FUNCTION_BLOCK FB_AUT_MODIFY EXTENDS FB_AUT_ABSTRACT
    (****************************************************************************)
    (*	POU_AUT_zxx			Bausteinaufrufe Station	zxx							*)
    (*	Status				ungetestet											*)
    (*  Version:			1.0													*)
    (*	Beschrieb:																*)
    (*																			*)
    (*	Abläufe:			FB_ABLzxxA		Hauptablauf							*)
    (*																			*)
    (*																			*)
    (* 	25.09.2019/Dj															*)
    (****************************************************************************)
    (*	dd.mm.yyyy   KZ    x.y			Beschrieb								*)
    (****************************************************************************)
VAR_INPUT
    (* spezifische Eingänge *)

END_VAR
VAR_OUTPUT
    (* spezifische Ausgänge *)

END_VAR
VAR
    (* Bausteine *)
    _FB_ABL_100A : FB_ABL_MODIFY;
END_VAR

(*******************************************************************)
(* Timer *)
(*******************************************************************)

(*******************************************************************)
(* Flanken / Merker *)
(*******************************************************************)
//MANU CYCLE
IF (enIN_State = StateMANU) AND xIN_ManuCycle THEN
    xManuCycle := TRUE;
END_IF;

IF (enIN_State <> StateMANU) OR xOUT_Done THEN
    xManuCycle := FALSE;
END_IF

//NEXT STEP
xNextStep := (enIN_State > StateSTEP) OR
             ((enIN_State = StateSTEP) AND xIN_Step) OR
             ((enIN_State = StateMANU) AND xManuCycle);

//RESET
xReset := ((enIN_State < StateREADY) AND (enIN_State <> StateINIT)) OR
          ((enIN_State = StateMANU) AND NOT xManuCycle);

(*******************************************************************)
(* Bausteinaufrufe Abläufe *)
(*******************************************************************)

_FB_ABL_100A(xIN_Reset       := xReset,
             xIN_Init        := xIN_Init,
             xIN_Quit        := xIN_Quit,
             xIN_Start       := enIN_State = enState.StateAUTO, //AND _FB_ABL_100A.xOUT_Done AND _FB_ABL_100A.xOUT_Ready,
             xIN_Sperre      := NOT xIN_On,
             xIN_NextStep    := xNextStep,
             xIN_AlarmAktiv  := xIN_AlarmAktiv,
             xIN_DryCycle    := xIN_DryCycle,
             xIN_RestartCYCL := enIN_State = enState.StateAUTO, // only restart when the mover has move out
             enIN_State      := enIN_State,
             tIN_Timeout     := tIN_Timeout,
             pxFG_Freigabe   := ADR(xDummy),
             Mover           := THIS^.Mover,
             xOUT_ErrFlag    =>,
             xOUT_Busy       =>,
             xOUT_Done       =>,
             xOUT_Timeout    =>,
             xOUT_InitDone   =>,
             xOUT_Wait       =>,
             iOUT_Step       =>,
             bOUT_Error      =>);
			 
(*******************************************************************)
(* Mover reset flags *)
(*******************************************************************)

(*******************************************************************)
(* OUTPUT *)
(*******************************************************************)
xOUT_InitDone := _FB_ABL_100A.xOUT_InitDone;
xOUT_Ready    := xOUT_InitDone;
xOUT_Done     := _FB_ABL_100A.xOUT_Done;
xOUT_ErrFlag  := _FB_ABL_100A.xOUT_ErrFlag;
xOUT_Wait     := _FB_ABL_100A.xOUT_Wait;
xOUT_AlarmST  := xOUT_ErrFlag;

(*******************************************************************)
(* Bausteinaufruf Error Station *)
(*******************************************************************)
// POU_ERR_VORLAGE(xIN_QUIT:=xIN_Quit , pstrArIN_ALARM:=ADR(HMI.strArALARM[1]));

METHOD GiveMover : IProcessSampleMover
VAR_INPUT
	mover : REFERENCE TO FB_Mover;
END_VAR
IF __ISVALIDREF(mover) THEN
    THIS^.Mover                       REF= mover;
END_IF
END_METHOD

(* % of completion of the process *)
PROPERTY iCompletionPC : INT
GET
iCompletionPC := THIS^._FB_ABL_100A.iOUT_ProcessCompletion;
END_GET
END_PROPERTY

(* Process time, expressed in milisecond *)
PROPERTY iProcessTimeMili : DINT
GET
iProcessTimeMili := TO_DINT(this^._FB_ABL_100A.iProcessTimeMili);
END_GET
SET
THIS^._FB_ABL_100A.iProcessTimeMili := TO_UDINT(iProcessTimeMili);
END_SET
END_PROPERTY

PROPERTY ProcessExecution : ProcessExecution_e
GET
ProcessExecution := THIS^._ProcessExecution;
END_GET
SET
THIS^._ProcessExecution := ProcessExecution;
END_SET
END_PROPERTY

METHOD TakeMover : IProcessSampleMover
VAR_INPUT
END_VAR
THIS^.Mover REF= 0;
END_METHOD

PROPERTY xBusy : BOOL
GET
xBusy := This^._FB_ABL_100A.xOUT_Busy;
END_GET
SET
END_SET
END_PROPERTY

PROPERTY xDone : BOOL
GET
xDone := THIS^._FB_ABL_100A.xOUT_Ready OR THIS^._FB_ABL_100A.xOUT_Done;
END_GET
END_PROPERTY

PROPERTY xMoverPathFree : BOOL
GET
xMoverPathFree := THIS^._FB_ABL_100A.xOUT_MoverFree OR THIS^._FB_ABL_100A.xOUT_Ready OR THIS^._FB_ABL_100A.xOUT_Done;
END_GET
END_PROPERTY

PROPERTY xMoverShouldLeave : BOOL
GET
xMoverShouldLeave := THIS^._FB_ABL_100A.iOUT_Step = ST100_Modify_e.SYNC_MOVER_LEAVE;
END_GET
END_PROPERTY

END_FUNCTION_BLOCK

(* stored: Version 1.1.0.1, ProductVersion 3.1.4024.6
   POU FB_AUT_MODIFY: Id {8dba9628-8cc4-42a6-92b5-7f87e0d812eb}, SpecialFunc None
   Method GiveMover: Id {4c146103-7ffe-45aa-9d54-074e277de283}
   Property iCompletionPC: Id {f2589b9c-4322-4bcc-8ec7-67d5086b786f}
   Get Get: Id {a2149bc6-8489-49f4-a1d7-531f9b7366d9}
   Property iProcessTimeMili: Id {9f1e3260-10ad-4f56-ba1f-45709124d7c3}
   Get Get: Id {6b411cd5-f3d8-4c85-9154-60d64e5d9840}
   Set Set: Id {6445fa35-8e05-4eff-b02e-33bf402f26e0}
   Property ProcessExecution: Id {22172c17-84f7-49e0-98f2-995ca83d491f}
   Get Get: Id {45d6e0d5-3c68-456d-b95a-e8efd8af0d57}
   Set Set: Id {6623b9f6-97ea-4a84-b348-f2e5282e90fd}
   Method TakeMover: Id {922d3a02-c6b2-4874-8cbe-c40a087d83ed}
   Property xBusy: Id {b162fbc6-d2f1-4618-a8ff-8e63306c2460}
   Get Get: Id {2e5d95e3-c60a-44d2-9223-656d419ea6ef}
   Set Set: Id {e720c6e2-8c0b-4538-989c-5330517681eb}
   Property xDone: Id {3e5d470c-9bd6-4ecf-bf99-c3500006dae5}
   Get Get: Id {c99e3841-5816-4493-821e-2aa023478d68}
   Property xMoverPathFree: Id {4470c49a-46aa-420a-b633-4c04ce41ba5e}
   Get Get: Id {4db5cc6f-3c16-42d7-beff-53243016db52}
   Property xMoverShouldLeave: Id {28a57ad5-3b2d-4e74-b73f-fc9049c11636}
   Get Get: Id {8d4dd82a-a4d5-4d07-adb7-9d6696bcb254} *)
